INTERFACE IEventHandler_OnExecutionFailed EXTENDS IEventHandlerBase

METHOD OnExecutionFailed
VAR_INPUT
    Message : T_MaxString;
END_VAR
END_METHOD

END_INTERFACE

(* stored: Version 1.1.0.1, ProductVersion 3.1.4024.3
   Itf IEventHandler_OnExecutionFailed: Id {74b8c4a1-fb31-444a-a331-482f563eae8d}
   Method OnExecutionFailed: Id {789a7f7b-0a73-0296-366d-785fe9e2d47e} *)
